SUBAPPLICATION Uebung_003a_AX (* DigitalInput_I1/_I2 auf DigitalOutput_Q1/_I2 - mit typed Subapp *)
  (* Standard: 61499-2; Description: Copyright (c) 2023 Meisterschulen am Ostbahnhof This program and the accompanying materials are made available under the terms of the Eclipse Public License 2.0 which is available at https://www.eclipse.org/legal/epl-2.0/ SPDX-License-Identifier: EPL-2.0 *)
  (* Version 1.0, 2023-10-23, Franz Höpfinger, Meisterschulen am Ostbahnhof *)
  PACKAGE Uebungen;
  IMPORT logiBUS::io::DI::logiBUS_DI::Input_I1;
  IMPORT logiBUS::io::DI::logiBUS_DI::Input_I2;
  IMPORT logiBUS::io::DQ::logiBUS_DO::Output_Q1;
  IMPORT logiBUS::io::DQ::logiBUS_DO::Output_Q2;
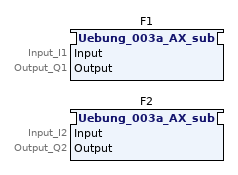
  SUBAPPS
    F1 : Uebungen::Uebung_003a_AX_sub(Input := Input_I1, Output := Output_Q1);
    F2 : Uebungen::Uebung_003a_AX_sub(Input := Input_I2, Output := Output_Q2);
  END_SUBAPPS
END_SUBAPPLICATION
